// Mitsubishi GX Works2 project: fistukUpdated_with_everyone   PLC: FX3G

// global labels: Global1
VAR_GLOBAL
  PowerOn AT X007 : BOOL;
  WorkDayLight AT Y007 : BOOL;
  Input1 AT D1140 : REAL;
  Nuts AT D1155 : REAL;
  Input2 AT D1160 : REAL;
  Fistuk AT D1165 : REAL;
  Input3 AT D1170 : REAL;
  Kadaif AT D1175 : REAL;
  FinishInput AT M5 : BOOL;
END_VAR
VAR_GLOBAL CONSTANT
  MinNuts : REAL := 100.0;
  MinFistuk : REAL := 120.0;
  MinKadaif : REAL := 60.0;
END_VAR
VAR_GLOBAL
  GoodNuts AT M10 : BOOL;
  GoodFistuk AT M15 : BOOL;
  GoodAll AT M20 : BOOL;
  NumArizot AT D1180 : INT;
  FinishDay AT M25 : BOOL;
  Sample AT Y006 : BOOL;
  Emergency AT X005 : BOOL;
  CheckLight AT Y000 : BOOL;
  Input4 AT D1180 : REAL;
  Chocklate AT D1185 : REAL;
END_VAR
VAR_GLOBAL CONSTANT
  MinChocklate : REAL := 400;
END_VAR
VAR_GLOBAL
  GoodChocklate AT M17 : BOOL;
  StartMelting AT X001 : BOOL;
  TemperatureSwitch AT X002 : BOOL;
  MeltingLight AT Y001 : BOOL;
  StartYezika AT M30 : BOOL;
  ReadtToStartYezika AT M30 : BOOL;
  ReadyToStartYezika AT M30 : BOOL;
  TavnitInPlace AT X003 : BOOL;
  PassedFourSec AT M35 : BOOL;
  Counter1 AT TC1 : BOOL;
END_VAR
VAR_GLOBAL CONSTANT
  Forty : WORD := 40;
END_VAR
VAR_GLOBAL
  YezikaOn AT Y002 : BOOL;
  TimeYezika AT TS1 : BOOL;
  ReadAnalog AT X004 : BOOL;
  AnalogInput1 AT D8280 : INT;
  InputAnalog AT D1200 : REAL;
END_VAR
VAR_GLOBAL CONSTANT
  ChooseNuts : REAL := 5;
END_VAR
VAR_GLOBAL
  NutsChosen AT M45 : BOOL;
  DubaiChosen AT M50 : BOOL;
END_VAR
VAR_GLOBAL CONSTANT
  ChooseDubai : REAL := 10;
END_VAR
VAR_GLOBAL
  Analog11 AT D1215 : INT;
END_VAR
VAR_GLOBAL CONSTANT
  Initiate : REAL := 400;
END_VAR
VAR_GLOBAL
  Temp1 AT D7755 : INT;
  SaveAnalog1 AT D8201 : REAL;
END_VAR
VAR_GLOBAL CONSTANT
  Inition : REAL := 400;
END_VAR
VAR_GLOBAL
  KeepAnalog AT D8201 : REAL;
END_VAR
VAR_GLOBAL CONSTANT
  NutsChoose : REAL := 5;
END_VAR
VAR_GLOBAL
  DidNutsChosen AT M50 : BOOL;
  KindChosen AT M55 : BOOL;
  GoodCheck AT M155 : BOOL;
END_VAR
VAR_GLOBAL CONSTANT
  M_1 : REAL := 100;
  M_2 : REAL := 20;
  M_3 : REAL := 120;
  M_4 : REAL := 60;
END_VAR
VAR_GLOBAL
  FinishChoosing AT M60 : BOOL;
  Counter2 AT TC2 : BOOL;
END_VAR
VAR_GLOBAL CONSTANT
  Fifty : WORD := 50;
END_VAR
VAR_GLOBAL
  TimeCream AT TS2 : BOOL;
  LightSwitch AT M65 : BOOL;
  Counter3 AT TC3 : BOOL;
END_VAR
VAR_GLOBAL CONSTANT
  Shtaim : WORD := 2;
END_VAR
VAR_GLOBAL
  TimeHivHuv AT TS3 : BOOL;
  HivLight AT Y003 : BOOL;
  HuvLight AT Y004 : BOOL;
  Counter4 AT TC4 : BOOL;
  TimeHivHuv2 AT TS4 : BOOL;
  SwitchEnded AT M70 : BOOL;
END_VAR
VAR_GLOBAL CONSTANT
  Hamesh : WORD := 5;
END_VAR
VAR_GLOBAL
  Colding AT X006 : BOOL;
  Counter5 AT TC5 : BOOL;
END_VAR
VAR_GLOBAL CONSTANT
  Shalosh : WORD := 30;
END_VAR
VAR_GLOBAL
  TimeY6 AT TS5 : BOOL;
  ColdingLight AT Y006 : BOOL;
  FinishTable AT X000 : BOOL;
  TableConter AT CC1 : BOOL;
  TableCounter AT CC9 : BOOL;
END_VAR
VAR_GLOBAL CONSTANT
  Conter7 : INT := 4;
END_VAR
VAR_GLOBAL
  NumTables AT CS1 : BOOL;
  NumFinish AT CS9 : BOOL;
END_VAR
VAR_GLOBAL CONSTANT
  ConsArizott : REAL := 1;
END_VAR
VAR_GLOBAL
  PackingLight AT Y005 : BOOL;
  UpdateAna AT M100 : BOOL;
END_VAR
VAR_GLOBAL CONSTANT
  Conter8 : INT := 1;
  Conter66 : INT := 4;
END_VAR
VAR_GLOBAL
  ArizotNum AT D1510 : REAL;
  ArizotNumDiv AT D1520 : REAL;
END_VAR
VAR_GLOBAL CONSTANT
  Conter666 : REAL := 4;
  FortyF : REAL := 40;
END_VAR
VAR_GLOBAL
  AnalogOutput AT D8282 : INT;
  StartFive AT M105 : BOOL;
  FhinishHivhuv AT TS2 : BOOL;
END_VAR
VAR_GLOBAL CONSTANT
  Ehad : WORD := 1;
  Conter6661 : REAL := 1;
END_VAR
VAR_GLOBAL
  StartSix AT M115 : BOOL;
  Hhhhhh AT M225 : BOOL;
  FhinishMana AT M135 : BOOL;
END_VAR

// task Task_01 (event TRUE, interval 0, priority 31): POU_01

PROGRAM POU_01
VAR
  kind_chosen : BOOL;
END_VAR
VAR CONSTANT
  Conter6 : WORD := 4;
END_VAR
(* structured ladder/FBD written out as ST: instructions are called as NAME(EN, inputs, outputs); _pN, _eN, _tN stand for wires *)
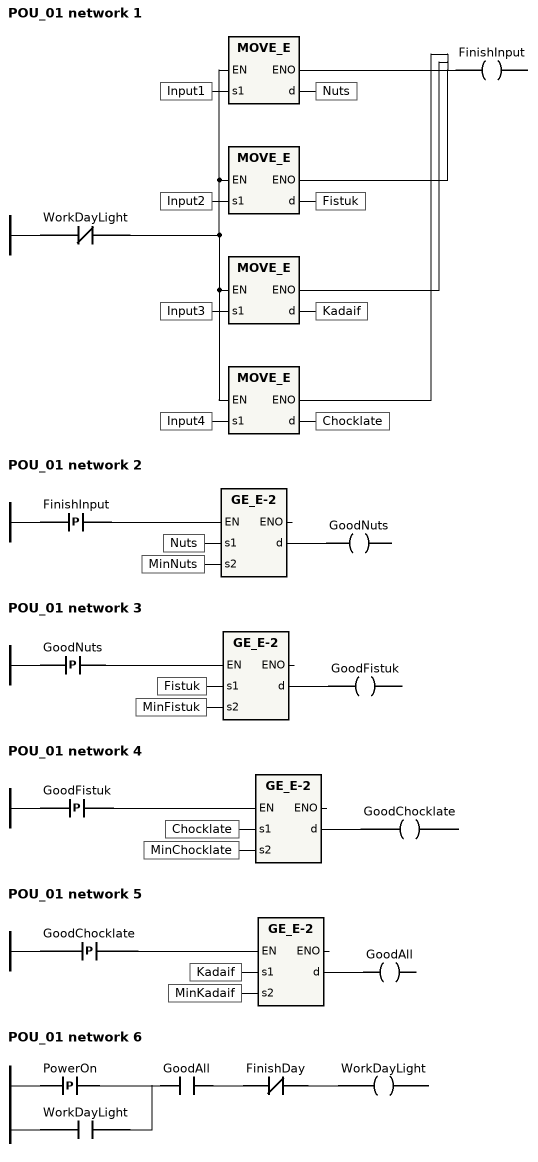
(* network 1 *)
_p1 := NOT WorkDayLight;
_e2 := MOVE_E(_p1, Input1, Nuts);
_e3 := MOVE_E(_p1, Input2, Fistuk);
_e4 := MOVE_E(_p1, Input3, Kadaif);
_e5 := MOVE_E(_p1, Input4, Chocklate);
FinishInput := _e2 OR _e3 OR _e4 OR _e5;
(* network 2 *)
GE_E(LDP(TRUE, FinishInput), Nuts, MinNuts, _t1);
GoodNuts := _t1;
(* network 3 *)
GE_E(LDP(TRUE, GoodNuts), Fistuk, MinFistuk, _t1);
GoodFistuk := _t1;
(* network 4 *)
GE_E(LDP(TRUE, GoodFistuk), Chocklate, MinChocklate, _t1);
GoodChocklate := _t1;
(* network 5 *)
GE_E(LDP(TRUE, GoodChocklate), Kadaif, MinKadaif, _t1);
GoodAll := _t1;
(* network 6 *)
WorkDayLight := ((LDP(TRUE, PowerOn) OR WorkDayLight) AND GoodAll) AND NOT FinishDay;
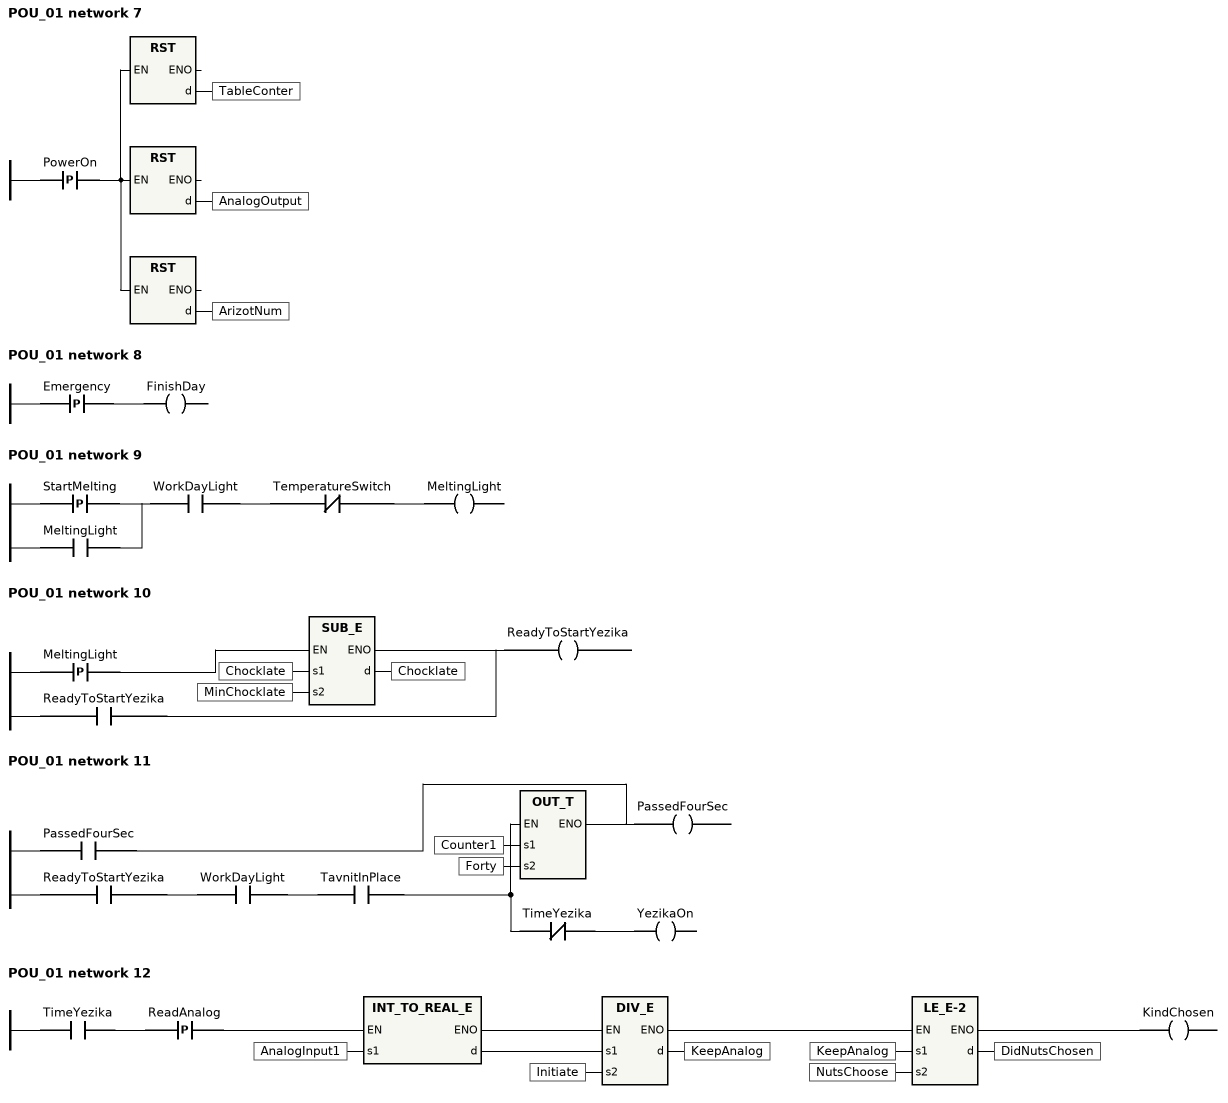
(* network 7 *)
_p1 := LDP(TRUE, PowerOn);
RST(_p1, TableConter);
RST(_p1, AnalogOutput);
RST(_p1, ArizotNum);
(* network 8 *)
FinishDay := LDP(TRUE, Emergency);
(* network 9 *)
MeltingLight := ((LDP(TRUE, StartMelting) OR MeltingLight) AND WorkDayLight) AND NOT TemperatureSwitch;
(* network 10 *)
_e1 := SUB_E(LDP(TRUE, MeltingLight), Chocklate, MinChocklate, Chocklate);
ReadyToStartYezika := _e1 OR ReadyToStartYezika;
(* network 11 *)
_p1 := ReadyToStartYezika AND WorkDayLight AND TavnitInPlace;
_e2 := OUT_T(_p1, Counter1, Forty);
PassedFourSec := PassedFourSec OR _e2;
YezikaOn := _p1 AND NOT TimeYezika;
(* network 12 *)
_e2 := INT_TO_REAL_E(TimeYezika AND LDP(TRUE, ReadAnalog), AnalogInput1, _t1);
_e3 := DIV_E(_e2, _t1, Initiate, KeepAnalog);
_e4 := LE_E(_e3, KeepAnalog, NutsChoose, DidNutsChosen);
KindChosen := _e4;
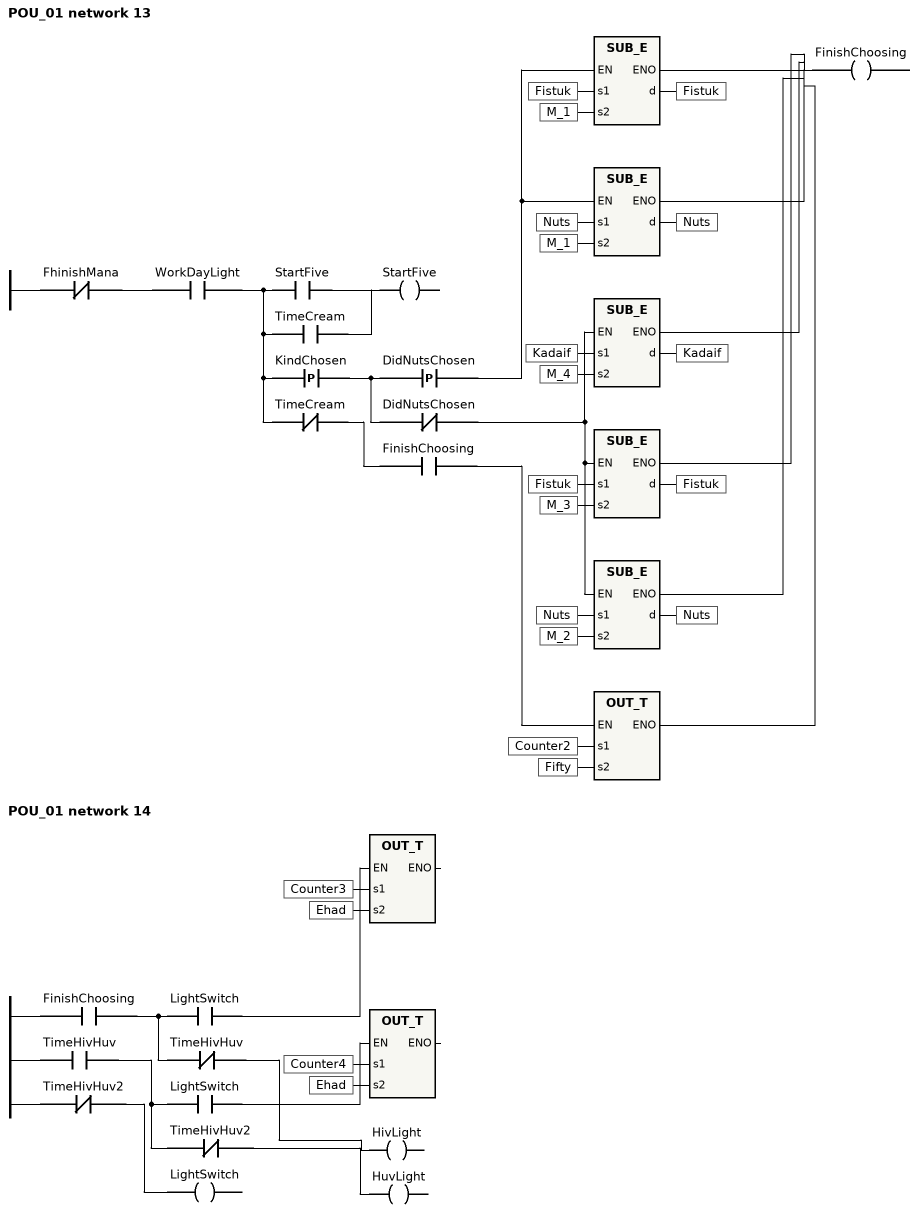
(* network 13 *)
_p1 := NOT FhinishMana AND WorkDayLight;
StartFive := (_p1 AND StartFive) OR (_p1 AND TimeCream);
_p2 := _p1 AND LDP(TRUE, KindChosen);
_p3 := _p2 AND LDP(TRUE, DidNutsChosen);
_e4 := SUB_E(_p3, Fistuk, M_1, Fistuk);
_e5 := SUB_E(_p3, Nuts, M_1, Nuts);
_p6 := _p2 AND NOT DidNutsChosen;
_e7 := SUB_E(_p6, Kadaif, M_4, Kadaif);
_e8 := SUB_E(_p6, Fistuk, M_3, Fistuk);
_e9 := SUB_E(_p6, Nuts, M_2, Nuts);
_e10 := OUT_T(_p1 AND NOT TimeCream AND FinishChoosing, Counter2, Fifty);
FinishChoosing := _e4 OR _e5 OR _e7 OR _e8 OR _e9 OR _e10;
(* network 14 *)
OUT_T(FinishChoosing AND LightSwitch, Counter3, Ehad);
HivLight := FinishChoosing AND NOT TimeHivHuv;
OUT_T(TimeHivHuv AND LightSwitch, Counter4, Ehad);
HuvLight := TimeHivHuv AND NOT TimeHivHuv2;
LightSwitch := NOT TimeHivHuv2;
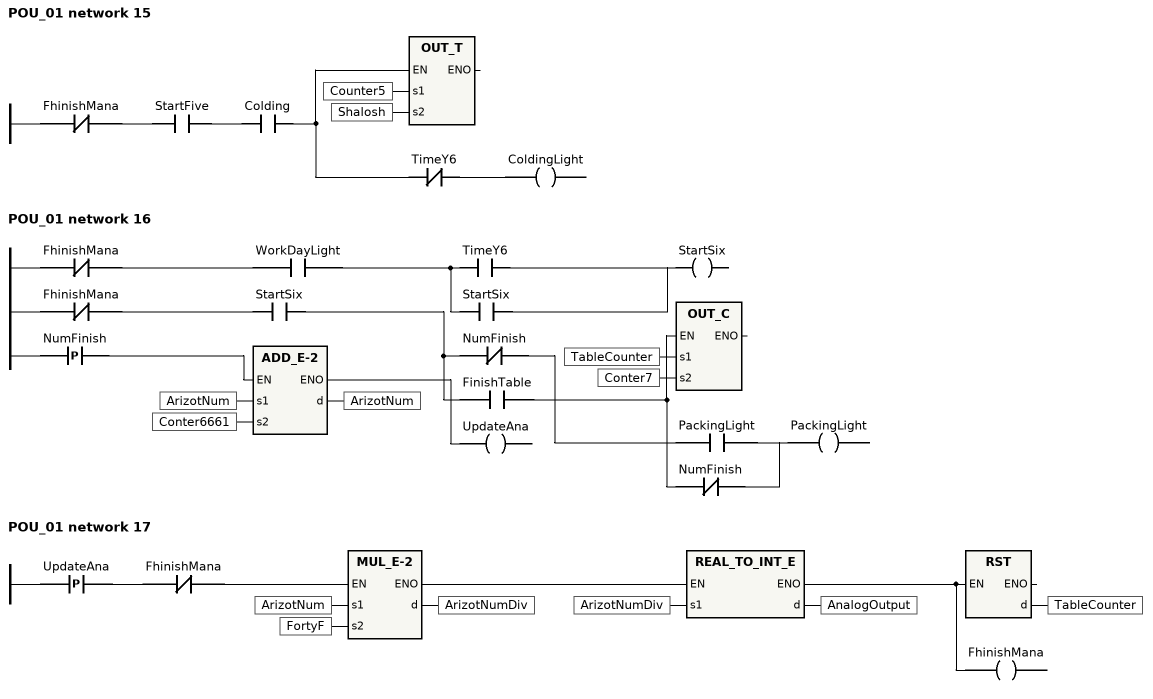
(* network 15 *)
_p1 := NOT FhinishMana AND StartFive AND Colding;
OUT_T(_p1, Counter5, Shalosh);
ColdingLight := _p1 AND NOT TimeY6;
(* network 16 *)
_p1 := NOT FhinishMana AND WorkDayLight;
StartSix := (_p1 AND TimeY6) OR (_p1 AND StartSix);
_p2 := NOT FhinishMana AND StartSix;
_p3 := _p2 AND FinishTable;
PackingLight := (_p2 AND NOT NumFinish AND PackingLight) OR (_p3 AND NOT NumFinish);
OUT_C(_p3, TableCounter, Conter7);
_e4 := ADD_E(LDP(TRUE, NumFinish), ArizotNum, Conter6661, ArizotNum);
UpdateAna := _e4;
(* network 17 *)
_e1 := MUL_E(LDP(TRUE, UpdateAna) AND NOT FhinishMana, ArizotNum, FortyF, ArizotNumDiv);
_e2 := REAL_TO_INT_E(_e1, ArizotNumDiv, AnalogOutput);
FhinishMana := _e2;
RST(_e2, TableCounter);
END_PROGRAM
